FUNCTION_BLOCK Mc3SlaveAxisPTP EXTENDS Mc3AxisPTP IMPLEMENTS I_Mc3SlaveAxis
VAR
	// Tasks
	MotionCoupleTaskGearing : Mc3MotionCoupleTask_Gearing := (Name := 'MC GearIn');
END_VAR

(*FB_Init is always available implicitly and it is used primarily for initialization.
The return value is not evaluated. For a specific influence, you can also declare the
methods explicitly and provide additional code there with the standard initialization
code. You can evaluate the return value.*)
METHOD FB_Init : BOOL
VAR_INPUT
	(* TRUE: the retain variables are initialized (reset warm / reset cold)*)
	bInitRetains : BOOL;

	(* TRUE: the instance will be copied to the copy code afterward (online change)   *)
	bInCopyCode : BOOL;
	Name		: T_MaxString;
	Axis		: REFERENCE TO Tc3_Mc3Ptp.AXIS_REF;
END_VAR
// Register all Motion Tasks to Collection
MotionTaskCollection.AddTask(MotionCoupleTaskGearing);
END_METHOD

METHOD GearIn
VAR_INPUT
END_VAR
MotionCoupleTaskGearing.GearIn	  := TRUE;
MotionCoupleTaskGearing.BufferMode := _McBufferMode;
MotionCoupleTaskGearing.Execute();
END_METHOD

METHOD GearOut
VAR_INPUT
END_VAR
MotionCoupleTaskGearing.GearIn := FALSE;
MotionCoupleTaskGearing.Execute();
END_METHOD

{attribute 'monitoring' := 'call'}
PROPERTY InGear : BOOL
GET
InGear := MotionCoupleTaskGearing.InGear;
END_GET
END_PROPERTY

PROPERTY Master : I_Mc3Axis
SET
MotionCoupleTaskGearing.Master := Master;
END_SET
END_PROPERTY

{attribute 'monitoring' := 'call'}
PROPERTY MasterHasError : BOOL
GET
MasterHasError := MotionCoupleTaskGearing.MasterHasError;
END_GET
END_PROPERTY

{attribute 'monitoring' := 'call'}
PROPERTY RatioDenominator : UDINT
SET
MotionCoupleTaskGearing.RatioDenominator := RatioDenominator;
END_SET
END_PROPERTY

{attribute 'monitoring' := 'call'}
PROPERTY RatioNumerator : UDINT
SET
MotionCoupleTaskGearing.RatioNumerator := RatioNumerator;
END_SET
END_PROPERTY

PROPERTY ReactionToMasterError : EReactionToMasterError
SET
MotionCoupleTaskGearing.ReactionToMasterError := ReactionToMasterError;
END_SET
END_PROPERTY

PROPERTY ReactionToSlaveError : EReactionToSlaveError
SET
MotionCoupleTaskGearing.ReactionToSlaveError := ReactionToSlaveError;
END_SET
END_PROPERTY

END_FUNCTION_BLOCK

(* stored: Version 1.1.0.1, ProductVersion 3.1.4026.20
   POU Mc3SlaveAxisPTP: Id {dbb109bb-ff39-4a6f-a087-981a1094ab33}, SpecialFunc None
   Folder Component: Id {2da04bb4-0deb-45c3-9e14-e3fcbadcef2c}
   Folder Slave: Id {3dae7c56-29a8-4dc3-881b-3d6d127c664e}
   Method FB_Init: Id {896379fe-3986-4612-a939-5d8be89c90f5}
   Method GearIn: Id {6aa1ef06-238c-4e9a-8e1e-027ba24268e8}
   Method GearOut: Id {0d80b130-7a9b-4a56-b26a-6822fc2070f2}
   Property InGear: Id {ef68c975-6eb7-4ab8-99a6-34db1f43f6b6}
   Get Get: Id {683a9448-ebcb-450c-bdd6-52fef9360173}
   Property Master: Id {f1287072-4640-4296-9c46-98f9bd407eb7}
   Set Set: Id {32fbebc8-3d35-4eb0-afa4-bba233fa4028}
   Property MasterHasError: Id {1d15a742-811f-48ee-aed2-db387a142c0c}
   Get Get: Id {aeedab01-befa-4f7b-959f-7a9c38243c0f}
   Property RatioDenominator: Id {260b178c-ac1e-4e92-bced-20a6ab9419f2}
   Set Set: Id {ffaf907e-180c-4dd0-8787-bf26522094bf}
   Property RatioNumerator: Id {aafc7b11-6fdc-49e9-8029-f6214fb9ccd8}
   Set Set: Id {251ba9a0-8610-4379-8a5e-9884753f2534}
   Property ReactionToMasterError: Id {1aa01e92-68b9-4003-a2e6-bf528bcecc07}
   Set Set: Id {8d4e56b3-cc5c-4e57-bba4-1db0decde057}
   Property ReactionToSlaveError: Id {f208a3bb-d78f-40af-bd74-d441b5d623ea}
   Set Set: Id {efeb8246-7c32-45ab-a4cf-964b1c73433e} *)
